// TIA Portal V17 export
// export: Created 2023-12-01T07:01:25.0311241Z, ExportSetting None, DisplayName Totally Integrated Automation Portal, DisplayVersion V17 Update 5, DisplayName TIA Portal Openness, DisplayVersion V17 Update 5, DisplayName TIA Portal Teamcenter Gateway, DisplayVersion V17 Update 5, DisplayName TIA Portal Version Control Interface, DisplayVersion V17, DisplayName SINAMICS Startdrive Advanced, DisplayVersion V17, DisplayName SINAMICS Startdrive G130, G150, S120, S150, SINAMICS MV, S210, DisplayVersion V17, DisplayName SINAMICS Startdrive G110M, G120, G120C, G120D, G120P, G115D, DisplayVersion V17, DisplayName STEP 7 Professional, DisplayVersion V17 Update 5, DisplayName STEP 7 Safety, DisplayVersion V17, DisplayName WinCC Advanced / Unified PC, DisplayVersion V17 Update 5
DATA_BLOCK "Blocco_dati_1"   // DB8
{ S7_Optimized_Access := 'TRUE' }
// stored: InstanceOfName EStrusore_OUT, InstanceOfType UDT
"EStrusore_OUT"
   // VAR
   //    MarciaDosatori : Bool;
   //    Allarme : Bool;
   //    bit_2 : Bool;
   //    bit_3 : Bool;
   //    bit_4 : Bool;
   //    bit_5 : Bool;
   //    bit_6 : Bool;
   //    bit_7 : Bool;
   //    bit_8 : Bool;
   //    bit_9 : Bool;
   //    bit_10 : Bool;
   //    bit_11 : Bool;
   //    bit_12 : Bool;
   //    bit_13 : Bool;
   //    bit_14 : Bool;
   //    bit_15 : Bool;
   // END_VAR
BEGIN
END_DATA_BLOCK
